//=============================================================================
// ST10_Flow8_FRobot_2.scl
// 1:1 CONVERSION FROM TIA PORTAL V18 GRAPH XML
// Generated: 2026-02-02
//=============================================================================

TYPE
    E_STEP_ST10_Flow8_FRobot_2 : (
        STEP_ST10_Flow8_FRobot_2_WaitRobotScanGripPos2Reach := 304,
        STEP_ST10_Flow8_FRobot_2_S2 := 2,
        STEP_ST10_Flow8_FRobot_2_Step380 := 380,
        STEP_ST10_Flow8_FRobot_2_CodeMove := 248,
        STEP_ST10_Flow8_FRobot_2_F8_Initial := 1,
        STEP_ST10_Flow8_FRobot_2_Maintenance_Pos := 850,
        STEP_ST10_Flow8_FRobot_2_WaitRobotScanGripPos4Reach := 383,
        STEP_ST10_Flow8_FRobot_2_PutPress := 145,
        STEP_ST10_Flow8_FRobot_2_PressGluePickProcessFinish := 549,
        STEP_ST10_Flow8_FRobot_2_WaitRobotScanGripPos3Reach := 372,
        STEP_ST10_Flow8_FRobot_2_DataMove_4 := 262,
        STEP_ST10_Flow8_FRobot_2_Brake_Test := 133,
        STEP_ST10_Flow8_FRobot_2_RobotScanGripPos2Comp := 371,
        STEP_ST10_Flow8_FRobot_2_WaitRobotGripStatus_2 := 366,
        STEP_ST10_Flow8_FRobot_2_S10_InitialFinish := 10,
        STEP_ST10_Flow8_FRobot_2_ScanNGPutFinish_1 := 349,
        STEP_ST10_Flow8_FRobot_2_GluePick := 140,
        STEP_ST10_Flow8_FRobot_2_S8 := 8,
        STEP_ST10_Flow8_FRobot_2_Data_Clear_2 := 258,
        STEP_ST10_Flow8_FRobot_2_WaitRobotFinish_3 := 353,
        STEP_ST10_Flow8_FRobot_2_S5_MESInitial := 5,
        STEP_ST10_Flow8_FRobot_2_DataMove_1 := 255,
        STEP_ST10_Flow8_FRobot_2_PickTableProcess := 400,
        STEP_ST10_Flow8_FRobot_2_StartRobotGlueNGPut := 344,
        STEP_ST10_Flow8_FRobot_2_PartOKStatus_1 := 269,
        STEP_ST10_Flow8_FRobot_2_StartRobotGluePut := 367,
        STEP_ST10_Flow8_FRobot_2_RobotAutoCycle := 329,
        STEP_ST10_Flow8_FRobot_2_BrakeTest_Req := 920,
        STEP_ST10_Flow8_FRobot_2_RobotStart := 316,
        STEP_ST10_Flow8_FRobot_2_GluePut := 155,
        STEP_ST10_Flow8_FRobot_2_PickPallet := 115,
        STEP_ST10_Flow8_FRobot_2_ScanNGPutProcess := 300,
        STEP_ST10_Flow8_FRobot_2_WaitRobot1AndRobot3HomeFinish := 379,
        STEP_ST10_Flow8_FRobot_2_WaitScanCompletely := 247,
        STEP_ST10_Flow8_FRobot_2_WaitRobotGripHaveStatus_3 := 354,
        STEP_ST10_Flow8_FRobot_2_Grip2PartStatus := 244,
        STEP_ST10_Flow8_FRobot_2_GlueNGPutProcess := 350,
        STEP_ST10_Flow8_FRobot_2_ScanMagane := 135,
        STEP_ST10_Flow8_FRobot_2_RobotHome := 317,
        STEP_ST10_Flow8_FRobot_2_WaitRobotGripHaveStatus_2 := 348,
        STEP_ST10_Flow8_FRobot_2_Open_NG_BOX_REQUESTED_ := 111,
        STEP_ST10_Flow8_FRobot_2_RobotScanGripPos4Comp := 391,
        STEP_ST10_Flow8_FRobot_2_Step930 := 930,
        STEP_ST10_Flow8_FRobot_2_ProcessStart := 100,
        STEP_ST10_Flow8_FRobot_2_WaitGripperPos3ScanFinish := 373,
        STEP_ST10_Flow8_FRobot_2_WaitGripperPos1ScanFinish := 296,
        STEP_ST10_Flow8_FRobot_2_WaitGripperPos4ScanFinish := 385,
        STEP_ST10_Flow8_FRobot_2_S_900 := 900,
        STEP_ST10_Flow8_FRobot_2_PartOKStatus := 249,
        STEP_ST10_Flow8_FRobot_2_WaitRobotFinish_1 := 343,
        STEP_ST10_Flow8_FRobot_2_WaitRobotGripStatus_3 := 369,
        STEP_ST10_Flow8_FRobot_2_Grip1PartStatus := 243,
        STEP_ST10_Flow8_FRobot_2_RobotScanGripPos1Comp := 301,
        STEP_ST10_Flow8_FRobot_2_StartRobotPutPress := 361,
        STEP_ST10_Flow8_FRobot_2_WaitRobotHomeRequest := 706,
        STEP_ST10_Flow8_FRobot_2_BrakeTestFinish := 929,
        STEP_ST10_Flow8_FRobot_2_S9 := 9,
        STEP_ST10_Flow8_FRobot_2_Tablecode_Scan := 200,
        STEP_ST10_Flow8_FRobot_2_StartRobotScanNGPut := 328,
        STEP_ST10_Flow8_FRobot_2_ScanMaganeProcess := 450,
        STEP_ST10_Flow8_FRobot_2_StartRobotPickPalletShaft := 326,
        STEP_ST10_Flow8_FRobot_2_WaitRobotFinish_4 := 356,
        STEP_ST10_Flow8_FRobot_2_DataMove_3 := 260,
        STEP_ST10_Flow8_FRobot_2_ScanMaganeProcessFinish := 499,
        STEP_ST10_Flow8_FRobot_2_ScanNGPut := 120,
        STEP_ST10_Flow8_FRobot_2_WaitRobotGripHaveStatus_1 := 347,
        STEP_ST10_Flow8_FRobot_2_DataMove_5 := 264,
        STEP_ST10_Flow8_FRobot_2_MES_Online__offline_ := 384,
        STEP_ST10_Flow8_FRobot_2_WaitRobotFinish_5 := 359,
        STEP_ST10_Flow8_FRobot_2_ScanStart := 246,
        STEP_ST10_Flow8_FRobot_2_PartNGStatus := 251,
        STEP_ST10_Flow8_FRobot_2_Gripe1StatusAlarm := 331,
        STEP_ST10_Flow8_FRobot_2_CheckScanReady := 245,
        STEP_ST10_Flow8_FRobot_2_Gripe2StatusAlarm := 332,
        STEP_ST10_Flow8_FRobot_2_ScanFixtureCode := 110,
        STEP_ST10_Flow8_FRobot_2_WaitRobotGripHaveStatus := 346,
        STEP_ST10_Flow8_FRobot_2_WaitRobotFinish_2 := 345,
        STEP_ST10_Flow8_FRobot_2_PutProcessFinish := 599,
        STEP_ST10_Flow8_FRobot_2_WaitR1HomePosFinsh_1 := 899,
        STEP_ST10_Flow8_FRobot_2_GlueNGPut := 125,
        STEP_ST10_Flow8_FRobot_2_DataMove := 253,
        STEP_ST10_Flow8_FRobot_2_Maintenance := 131,
        STEP_ST10_Flow8_FRobot_2_GluePickProcess := 500,
        STEP_ST10_Flow8_FRobot_2_SetGripCodeScanFlag := 336,
        STEP_ST10_Flow8_FRobot_2_ReqRobotToMantenPos_1 := 704,
        STEP_ST10_Flow8_FRobot_2_WaitRobotReachScanPos := 357,
        STEP_ST10_Flow8_FRobot_2_GlueNGPutFinish := 399,
        STEP_ST10_Flow8_FRobot_2_PickTableProcessFinish := 449,
        STEP_ST10_Flow8_FRobot_2_MasteringTest_Req := 910,
        STEP_ST10_Flow8_FRobot_2_StartRobotScanGripperCode := 338,
        STEP_ST10_Flow8_FRobot_2_RobotScanGripperReachPos1 := 340,
        STEP_ST10_Flow8_FRobot_2_WaitMasteringTestFinish := 911,
        STEP_ST10_Flow8_FRobot_2_WaitRobotGripStatus := 360,
        STEP_ST10_Flow8_FRobot_2_S3 := 3,
        STEP_ST10_Flow8_FRobot_2_PickPalletFinish := 299,
        STEP_ST10_Flow8_FRobot_2_PutPressProcess := 550,
        STEP_ST10_Flow8_FRobot_2_Grip1SensorError := 266,
        STEP_ST10_Flow8_FRobot_2_PressPickProcess := 600,
        STEP_ST10_Flow8_FRobot_2_Data_Clear_6 := 265,
        STEP_ST10_Flow8_FRobot_2_StartRobotScanRing := 355,
        STEP_ST10_Flow8_FRobot_2_WaitRobotFinish := 327,
        STEP_ST10_Flow8_FRobot_2_RobotTaskSelect := 333,
        STEP_ST10_Flow8_FRobot_2_Tablecode_ScanFinish := 149,
        STEP_ST10_Flow8_FRobot_2_GripStatusCheck := 330,
        STEP_ST10_Flow8_FRobot_2_WaitRobotFinish_8 := 368,
        STEP_ST10_Flow8_FRobot_2_WaitRobotFinish_7 := 365,
        STEP_ST10_Flow8_FRobot_2_StartRobotPressPick := 364,
        STEP_ST10_Flow8_FRobot_2_WaitR1MaintenPosFinsh_1 := 705,
        STEP_ST10_Flow8_FRobot_2_PickTable := 130,
        STEP_ST10_Flow8_FRobot_2_RobotReady_ := 311,
        STEP_ST10_Flow8_FRobot_2_Masref_test := 132,
        STEP_ST10_Flow8_FRobot_2_GluePutProcess := 650,
        STEP_ST10_Flow8_FRobot_2_StartRobotGluePick := 358,
        STEP_ST10_Flow8_FRobot_2_PressPickProcessFinish_ := 649,
        STEP_ST10_Flow8_FRobot_2_ReqRobotToHomePos := 707,
        STEP_ST10_Flow8_FRobot_2_DataClear := 252,
        STEP_ST10_Flow8_FRobot_2_StartRobotPickTable := 352,
        STEP_ST10_Flow8_FRobot_2_WaitRobotStartHome := 381,
        STEP_ST10_Flow8_FRobot_2_GluePutProcessFinish := 699,
        STEP_ST10_Flow8_FRobot_2_WaitRobotGripStatus_1 := 363,
        STEP_ST10_Flow8_FRobot_2_WaitRobotFinish_6 := 362,
        STEP_ST10_Flow8_FRobot_2_PickPalletProcess := 250,
        STEP_ST10_Flow8_FRobot_2_RobotSpeed := 4,
        STEP_ST10_Flow8_FRobot_2_RobotManuallyMoved_ := 382,
        STEP_ST10_Flow8_FRobot_2_DataMove_2 := 257,
        STEP_ST10_Flow8_FRobot_2_Grip2SensorError := 267,
        STEP_ST10_Flow8_FRobot_2_WaitBrakeTestFinish := 921,
        STEP_ST10_Flow8_FRobot_2_FlagReset := 268,
        STEP_ST10_Flow8_FRobot_2_PressPick := 150,
        STEP_ST10_Flow8_FRobot_2_WaitGripperPos2ScanFinish := 337,
        STEP_ST10_Flow8_FRobot_2_RobotScanGripPos3Comp := 378,
        STEP_ST10_Flow8_FRobot_2_MasteringTestFinish := 919,
    ) INT := 1;
END_TYPE

CONST
    STEP_ST10_Flow8_FRobot_2_WaitRobotScanGripPos2Reach := 304;
    STEP_ST10_Flow8_FRobot_2_S2 := 2;
    STEP_ST10_Flow8_FRobot_2_Step380 := 380;
    STEP_ST10_Flow8_FRobot_2_CodeMove := 248;
    STEP_ST10_Flow8_FRobot_2_F8_Initial := 1;
    STEP_ST10_Flow8_FRobot_2_Maintenance_Pos := 850;
    STEP_ST10_Flow8_FRobot_2_WaitRobotScanGripPos4Reach := 383;
    STEP_ST10_Flow8_FRobot_2_PutPress := 145;
    STEP_ST10_Flow8_FRobot_2_PressGluePickProcessFinish := 549;
    STEP_ST10_Flow8_FRobot_2_WaitRobotScanGripPos3Reach := 372;
    STEP_ST10_Flow8_FRobot_2_DataMove_4 := 262;
    STEP_ST10_Flow8_FRobot_2_Brake_Test := 133;
    STEP_ST10_Flow8_FRobot_2_RobotScanGripPos2Comp := 371;
    STEP_ST10_Flow8_FRobot_2_WaitRobotGripStatus_2 := 366;
    STEP_ST10_Flow8_FRobot_2_S10_InitialFinish := 10;
    STEP_ST10_Flow8_FRobot_2_ScanNGPutFinish_1 := 349;
    STEP_ST10_Flow8_FRobot_2_GluePick := 140;
    STEP_ST10_Flow8_FRobot_2_S8 := 8;
    STEP_ST10_Flow8_FRobot_2_Data_Clear_2 := 258;
    STEP_ST10_Flow8_FRobot_2_WaitRobotFinish_3 := 353;
    STEP_ST10_Flow8_FRobot_2_S5_MESInitial := 5;
    STEP_ST10_Flow8_FRobot_2_DataMove_1 := 255;
    STEP_ST10_Flow8_FRobot_2_PickTableProcess := 400;
    STEP_ST10_Flow8_FRobot_2_StartRobotGlueNGPut := 344;
    STEP_ST10_Flow8_FRobot_2_PartOKStatus_1 := 269;
    STEP_ST10_Flow8_FRobot_2_StartRobotGluePut := 367;
    STEP_ST10_Flow8_FRobot_2_RobotAutoCycle := 329;
    STEP_ST10_Flow8_FRobot_2_BrakeTest_Req := 920;
    STEP_ST10_Flow8_FRobot_2_RobotStart := 316;
    STEP_ST10_Flow8_FRobot_2_GluePut := 155;
    STEP_ST10_Flow8_FRobot_2_PickPallet := 115;
    STEP_ST10_Flow8_FRobot_2_ScanNGPutProcess := 300;
    STEP_ST10_Flow8_FRobot_2_WaitRobot1AndRobot3HomeFinish := 379;
    STEP_ST10_Flow8_FRobot_2_WaitScanCompletely := 247;
    STEP_ST10_Flow8_FRobot_2_WaitRobotGripHaveStatus_3 := 354;
    STEP_ST10_Flow8_FRobot_2_Grip2PartStatus := 244;
    STEP_ST10_Flow8_FRobot_2_GlueNGPutProcess := 350;
    STEP_ST10_Flow8_FRobot_2_ScanMagane := 135;
    STEP_ST10_Flow8_FRobot_2_RobotHome := 317;
    STEP_ST10_Flow8_FRobot_2_WaitRobotGripHaveStatus_2 := 348;
    STEP_ST10_Flow8_FRobot_2_Open_NG_BOX_REQUESTED_ := 111;
    STEP_ST10_Flow8_FRobot_2_RobotScanGripPos4Comp := 391;
    STEP_ST10_Flow8_FRobot_2_Step930 := 930;
    STEP_ST10_Flow8_FRobot_2_ProcessStart := 100;
    STEP_ST10_Flow8_FRobot_2_WaitGripperPos3ScanFinish := 373;
    STEP_ST10_Flow8_FRobot_2_WaitGripperPos1ScanFinish := 296;
    STEP_ST10_Flow8_FRobot_2_WaitGripperPos4ScanFinish := 385;
    STEP_ST10_Flow8_FRobot_2_S_900 := 900;
    STEP_ST10_Flow8_FRobot_2_PartOKStatus := 249;
    STEP_ST10_Flow8_FRobot_2_WaitRobotFinish_1 := 343;
    STEP_ST10_Flow8_FRobot_2_WaitRobotGripStatus_3 := 369;
    STEP_ST10_Flow8_FRobot_2_Grip1PartStatus := 243;
    STEP_ST10_Flow8_FRobot_2_RobotScanGripPos1Comp := 301;
    STEP_ST10_Flow8_FRobot_2_StartRobotPutPress := 361;
    STEP_ST10_Flow8_FRobot_2_WaitRobotHomeRequest := 706;
    STEP_ST10_Flow8_FRobot_2_BrakeTestFinish := 929;
    STEP_ST10_Flow8_FRobot_2_S9 := 9;
    STEP_ST10_Flow8_FRobot_2_Tablecode_Scan := 200;
    STEP_ST10_Flow8_FRobot_2_StartRobotScanNGPut := 328;
    STEP_ST10_Flow8_FRobot_2_ScanMaganeProcess := 450;
    STEP_ST10_Flow8_FRobot_2_StartRobotPickPalletShaft := 326;
    STEP_ST10_Flow8_FRobot_2_WaitRobotFinish_4 := 356;
    STEP_ST10_Flow8_FRobot_2_DataMove_3 := 260;
    STEP_ST10_Flow8_FRobot_2_ScanMaganeProcessFinish := 499;
    STEP_ST10_Flow8_FRobot_2_ScanNGPut := 120;
    STEP_ST10_Flow8_FRobot_2_WaitRobotGripHaveStatus_1 := 347;
    STEP_ST10_Flow8_FRobot_2_DataMove_5 := 264;
    STEP_ST10_Flow8_FRobot_2_MES_Online__offline_ := 384;
    STEP_ST10_Flow8_FRobot_2_WaitRobotFinish_5 := 359;
    STEP_ST10_Flow8_FRobot_2_ScanStart := 246;
    STEP_ST10_Flow8_FRobot_2_PartNGStatus := 251;
    STEP_ST10_Flow8_FRobot_2_Gripe1StatusAlarm := 331;
    STEP_ST10_Flow8_FRobot_2_CheckScanReady := 245;
    STEP_ST10_Flow8_FRobot_2_Gripe2StatusAlarm := 332;
    STEP_ST10_Flow8_FRobot_2_ScanFixtureCode := 110;
    STEP_ST10_Flow8_FRobot_2_WaitRobotGripHaveStatus := 346;
    STEP_ST10_Flow8_FRobot_2_WaitRobotFinish_2 := 345;
    STEP_ST10_Flow8_FRobot_2_PutProcessFinish := 599;
    STEP_ST10_Flow8_FRobot_2_WaitR1HomePosFinsh_1 := 899;
    STEP_ST10_Flow8_FRobot_2_GlueNGPut := 125;
    STEP_ST10_Flow8_FRobot_2_DataMove := 253;
    STEP_ST10_Flow8_FRobot_2_Maintenance := 131;
    STEP_ST10_Flow8_FRobot_2_GluePickProcess := 500;
    STEP_ST10_Flow8_FRobot_2_SetGripCodeScanFlag := 336;
    STEP_ST10_Flow8_FRobot_2_ReqRobotToMantenPos_1 := 704;
    STEP_ST10_Flow8_FRobot_2_WaitRobotReachScanPos := 357;
    STEP_ST10_Flow8_FRobot_2_GlueNGPutFinish := 399;
    STEP_ST10_Flow8_FRobot_2_PickTableProcessFinish := 449;
    STEP_ST10_Flow8_FRobot_2_MasteringTest_Req := 910;
    STEP_ST10_Flow8_FRobot_2_StartRobotScanGripperCode := 338;
    STEP_ST10_Flow8_FRobot_2_RobotScanGripperReachPos1 := 340;
    STEP_ST10_Flow8_FRobot_2_WaitMasteringTestFinish := 911;
    STEP_ST10_Flow8_FRobot_2_WaitRobotGripStatus := 360;
    STEP_ST10_Flow8_FRobot_2_S3 := 3;
    STEP_ST10_Flow8_FRobot_2_PickPalletFinish := 299;
    STEP_ST10_Flow8_FRobot_2_PutPressProcess := 550;
    STEP_ST10_Flow8_FRobot_2_Grip1SensorError := 266;
    STEP_ST10_Flow8_FRobot_2_PressPickProcess := 600;
    STEP_ST10_Flow8_FRobot_2_Data_Clear_6 := 265;
    STEP_ST10_Flow8_FRobot_2_StartRobotScanRing := 355;
    STEP_ST10_Flow8_FRobot_2_WaitRobotFinish := 327;
    STEP_ST10_Flow8_FRobot_2_RobotTaskSelect := 333;
    STEP_ST10_Flow8_FRobot_2_Tablecode_ScanFinish := 149;
    STEP_ST10_Flow8_FRobot_2_GripStatusCheck := 330;
    STEP_ST10_Flow8_FRobot_2_WaitRobotFinish_8 := 368;
    STEP_ST10_Flow8_FRobot_2_WaitRobotFinish_7 := 365;
    STEP_ST10_Flow8_FRobot_2_StartRobotPressPick := 364;
    STEP_ST10_Flow8_FRobot_2_WaitR1MaintenPosFinsh_1 := 705;
    STEP_ST10_Flow8_FRobot_2_PickTable := 130;
    STEP_ST10_Flow8_FRobot_2_RobotReady_ := 311;
    STEP_ST10_Flow8_FRobot_2_Masref_test := 132;
    STEP_ST10_Flow8_FRobot_2_GluePutProcess := 650;
    STEP_ST10_Flow8_FRobot_2_StartRobotGluePick := 358;
    STEP_ST10_Flow8_FRobot_2_PressPickProcessFinish_ := 649;
    STEP_ST10_Flow8_FRobot_2_ReqRobotToHomePos := 707;
    STEP_ST10_Flow8_FRobot_2_DataClear := 252;
    STEP_ST10_Flow8_FRobot_2_StartRobotPickTable := 352;
    STEP_ST10_Flow8_FRobot_2_WaitRobotStartHome := 381;
    STEP_ST10_Flow8_FRobot_2_GluePutProcessFinish := 699;
    STEP_ST10_Flow8_FRobot_2_WaitRobotGripStatus_1 := 363;
    STEP_ST10_Flow8_FRobot_2_WaitRobotFinish_6 := 362;
    STEP_ST10_Flow8_FRobot_2_PickPalletProcess := 250;
    STEP_ST10_Flow8_FRobot_2_RobotSpeed := 4;
    STEP_ST10_Flow8_FRobot_2_RobotManuallyMoved_ := 382;
    STEP_ST10_Flow8_FRobot_2_DataMove_2 := 257;
    STEP_ST10_Flow8_FRobot_2_Grip2SensorError := 267;
    STEP_ST10_Flow8_FRobot_2_WaitBrakeTestFinish := 921;
    STEP_ST10_Flow8_FRobot_2_FlagReset := 268;
    STEP_ST10_Flow8_FRobot_2_PressPick := 150;
    STEP_ST10_Flow8_FRobot_2_WaitGripperPos2ScanFinish := 337;
    STEP_ST10_Flow8_FRobot_2_RobotScanGripPos3Comp := 378;
    STEP_ST10_Flow8_FRobot_2_MasteringTestFinish := 919;
END_CONST

FUNCTION_BLOCK "ST10_Flow8_FRobot_2_1to1"
{ S7_Optimized_Access := 'TRUE' }
VERSION : 1.0

VAR_INPUT
    iSysInface : "RCS_SysComInterface_V1";
END_VAR

VAR_IN_OUT
    ioPM_Inface : "RCS_PMInterface_V1";
    ioStatus : Int;
END_VAR

VAR_OUTPUT
    oAlarmID : Int;
END_VAR

VAR
    State : INT := 1;
    act_InitialRun : Bool;
    act_InitialOK : Bool;
    act_WaitRunning : Bool;
    act_Running : Bool;
    act_ProcessComplete : Bool;
    act_ProcessStart : Bool;
    act_UnPause : Bool;
    bError : Bool;
    wErrorID : Word;
END_VAR

BEGIN
    //======================================================================
    // STATE MACHINE - Inline Transition Conditions
    //======================================================================

    CASE #State OF

        // ===========================================
        // STEP 304: WaitRobotScanGripPos2Reach
        // ===========================================
        STEP_ST10_Flow8_FRobot_2_WaitRobotScanGripPos2Reach:
            // No actions in XML

            // Transition to next step: 2
            IF TRUE THEN  // Sequential transition - review XML for actual condition
                #State := STEP_ST10_Flow8_FRobot_2_S2;
            END_IF;

        // ===========================================
        // STEP 2: S2
        // ===========================================
        STEP_ST10_Flow8_FRobot_2_S2:
            // No actions in XML

            // Transition to next step: 380
            IF TRUE THEN  // Sequential transition - review XML for actual condition
                #State := STEP_ST10_Flow8_FRobot_2_Step380;
            END_IF;

        // ===========================================
        // STEP 380: Step380
        // ===========================================
        STEP_ST10_Flow8_FRobot_2_Step380:
            // No actions in XML

            // Transition to next step: 248
            IF TRUE THEN  // Sequential transition - review XML for actual condition
                #State := STEP_ST10_Flow8_FRobot_2_CodeMove;
            END_IF;

        // ===========================================
        // STEP 248: CodeMove
        // ===========================================
        STEP_ST10_Flow8_FRobot_2_CodeMove:
            // Action Qualifier=N
            // Token: "AutoProcessData".F_Robot2Grip2.Code_1 := "KeyenceSR1000Ctrl_806A1DB".sHMI.Status.CurrentCode
            "AutoProcessData".F_Robot2Grip2.Code_1 := "KeyenceSR1000Ctrl_806A1DB".sHMI.Status.CurrentCode;

            // Transition to next step: 1
            IF TRUE THEN  // Sequential transition - review XML for actual condition
                #State := STEP_ST10_Flow8_FRobot_2_F8_Initial;
            END_IF;

        // ===========================================
        // STEP 1: F8_Initial
        // ===========================================
        STEP_ST10_Flow8_FRobot_2_F8_Initial:
            // Action Qualifier=S
            // Token: #ioPM_Inface.InitialRun
            #ioPM_Inface.InitialRun := TRUE;
            // Action Qualifier=R
            // Token: #ioPM_Inface.InitialOK
            #ioPM_Inface.InitialOK := FALSE;
            // Action Qualifier=R
            // Token: #ioPM_Inface.WaitRunning
            #ioPM_Inface.WaitRunning := FALSE;
            // Action Qualifier=R
            // Token: #ioPM_Inface.Running
            #ioPM_Inface.Running := FALSE;
            // Action Qualifier=R
            // Token: #ioPM_Inface.UnPause
            #ioPM_Inface.UnPause := FALSE;
            // Action Qualifier=R
            // Token: "Station_Sys".Cmd.Calibration
            "Station_Sys".Cmd.Calibration := FALSE;
            // Action Qualifier=R
            // Token: "Station_Sys".Cmd.ChangeOver
            "Station_Sys".Cmd.ChangeOver := FALSE;
            // Action Qualifier=N
            // Token: //"ST350_Sys".Cmd.DryRun
            //"ST350_Sys".Cmd.DryRun;
            // Action Qualifier=R
            // Token: "Station_Sys".Cmd.Reserve
            "Station_Sys".Cmd.Reserve := FALSE;
            // Action Qualifier=R
            // Token: "Station_Sys".Cmd.OneCycle
            "Station_Sys".Cmd.OneCycle := FALSE;
            // Action Qualifier=R
            // Token: "AutoProcessControl".Robot_2.PalletPickFlag
            "AutoProcessControl".Robot_2.PalletPickFlag := FALSE;
            // Action Qualifier=R
            // Token: "AutoProcessControl".Robot_2.MagnetScanFlag
            "AutoProcessControl".Robot_2.MagnetScanFlag := FALSE;
            // Action Qualifier=R
            // Token: "AutoProcessControl".Robot_2.GluePutFlag
            "AutoProcessControl".Robot_2.GluePutFlag := FALSE;
            // Action Qualifier=R
            // Token: "AutoProcessControl".Robot_2.GluePickFlag
            "AutoProcessControl".Robot_2.GluePickFlag := FALSE;
            // Action Qualifier=R
            // Token: "AutoProcessControl".Robot_2.Press2PutFlag
            "AutoProcessControl".Robot_2.Press2PutFlag := FALSE;
            // Action Qualifier=R
            // Token: "AutoProcessControl".Robot_2.GlueNGPutFlag
            "AutoProcessControl".Robot_2.GlueNGPutFlag := FALSE;
            // Action Qualifier=R
            // Token: "AutoProcessControl".Robot_2.ScanNGPutFlag
            "AutoProcessControl".Robot_2.ScanNGPutFlag := FALSE;
            // Action Qualifier=R
            // Token: #ioPM_Inface.ProcessComplete
            #ioPM_Inface.ProcessComplete := FALSE;
            // Action Qualifier=R
            // Token: #ioPM_Inface.ProcessStart
            #ioPM_Inface.ProcessStart := FALSE;
            // Action Qualifier=R
            // Token: "ChangeOver_DB".Robot_2.MaintenancePosReqSelFlag
            "ChangeOver_DB".Robot_2.MaintenancePosReqSelFlag := FALSE;
            // Action Qualifier=N
            // Token: //"Robot_DB".Robot_2.MasteringTest_Req
            //"Robot_DB".Robot_2.MasteringTest_Req;
            // Action Qualifier=N
            // Token: //"Robot_DB".Robot_2.BrakeTest_Req
            //"Robot_DB".Robot_2.BrakeTest_Req;
            // Action Qualifier=R
            // Token: #Auto_Run_after_NG_box_closed
            #Auto_Run_after_NG_box_closed := FALSE;

            // Transition to next step: 850
            IF TRUE THEN  // Sequential transition - review XML for actual condition
                #State := STEP_ST10_Flow8_FRobot_2_Maintenance_Pos;
            END_IF;

        // ===========================================
        // STEP 850: Maintenance Pos
        // ===========================================
        STEP_ST10_Flow8_FRobot_2_Maintenance_Pos:
            // No actions in XML

            // Transition to next step: 383
            IF TRUE THEN  // Sequential transition - review XML for actual condition
                #State := STEP_ST10_Flow8_FRobot_2_WaitRobotScanGripPos4Reach;
            END_IF;

        // ===========================================
        // STEP 383: WaitRobotScanGripPos4Reach
        // ===========================================
        STEP_ST10_Flow8_FRobot_2_WaitRobotScanGripPos4Reach:
            // No actions in XML

            // Transition to next step: 145
            IF TRUE THEN  // Sequential transition - review XML for actual condition
                #State := STEP_ST10_Flow8_FRobot_2_PutPress;
            END_IF;

        // ===========================================
        // STEP 145: PutPress
        // ===========================================
        STEP_ST10_Flow8_FRobot_2_PutPress:
            // Action Qualifier=S
            // Token: "AutoProcessControl".Robot_2.Press2PutFlag
            "AutoProcessControl".Robot_2.Press2PutFlag := TRUE;
            // Action Qualifier=R
            // Token: #ioPM_Inface.ProcessComplete
            #ioPM_Inface.ProcessComplete := FALSE;
            // Action Qualifier=S
            // Token: #ioPM_Inface.ProcessStart
            #ioPM_Inface.ProcessStart := TRUE;

            // Transition to next step: 549
            IF TRUE THEN  // Sequential transition - review XML for actual condition
                #State := STEP_ST10_Flow8_FRobot_2_PressGluePickProcessFinish;
            END_IF;

        // ===========================================
        // STEP 549: PressGluePickProcessFinish
        // ===========================================
        STEP_ST10_Flow8_FRobot_2_PressGluePickProcessFinish:
            // Action Qualifier=S
            // Token: #ioPM_Inface.ProcessComplete
            #ioPM_Inface.ProcessComplete := TRUE;
            // Action Qualifier=R
            // Token: #ioPM_Inface.ProcessStart
            #ioPM_Inface.ProcessStart := FALSE;

            // Transition to next step: 372
            IF TRUE THEN  // Sequential transition - review XML for actual condition
                #State := STEP_ST10_Flow8_FRobot_2_WaitRobotScanGripPos3Reach;
            END_IF;

        // ===========================================
        // STEP 372: WaitRobotScanGripPos3Reach
        // ===========================================
        STEP_ST10_Flow8_FRobot_2_WaitRobotScanGripPos3Reach:
            // No actions in XML

            // Transition to next step: 262
            IF TRUE THEN  // Sequential transition - review XML for actual condition
                #State := STEP_ST10_Flow8_FRobot_2_DataMove_4;
            END_IF;

        // ===========================================
        // STEP 262: DataMove_4
        // ===========================================
        STEP_ST10_Flow8_FRobot_2_DataMove_4:
            // Action Qualifier=N, Event="S1"
            // Token: "AutoProcessData".F_Robot2Grip1 := "AutoProcessData".B_Press1
            "AutoProcessData".F_Robot2Grip1 := "AutoProcessData".B_Press1;
            // Action Qualifier=N, Event="S1"
            // Token: "AutoProcessData".B_Press1 := "AutoProcessData".ClearData
            "AutoProcessData".B_Press1 := "AutoProcessData".ClearData;

            // Transition to next step: 133
            IF TRUE THEN  // Sequential transition - review XML for actual condition
                #State := STEP_ST10_Flow8_FRobot_2_Brake_Test;
            END_IF;

        // ===========================================
        // STEP 133: Brake_Test
        // ===========================================
        STEP_ST10_Flow8_FRobot_2_Brake_Test:
            // Action Qualifier=R
            // Token: #ioPM_Inface.ProcessComplete
            #ioPM_Inface.ProcessComplete := FALSE;
            // Action Qualifier=S
            // Token: #ioPM_Inface.ProcessStart
            #ioPM_Inface.ProcessStart := TRUE;

            // Transition to next step: 371
            IF TRUE THEN  // Sequential transition - review XML for actual condition
                #State := STEP_ST10_Flow8_FRobot_2_RobotScanGripPos2Comp;
            END_IF;

        // ===========================================
        // STEP 371: RobotScanGripPos2Comp
        // ===========================================
        STEP_ST10_Flow8_FRobot_2_RobotScanGripPos2Comp:
            // No actions in XML

            // Transition to next step: 366
            IF TRUE THEN  // Sequential transition - review XML for actual condition
                #State := STEP_ST10_Flow8_FRobot_2_WaitRobotGripStatus_2;
            END_IF;

        // ===========================================
        // STEP 366: WaitRobotGripStatus_2
        // ===========================================
        STEP_ST10_Flow8_FRobot_2_WaitRobotGripStatus_2:
            // No actions in XML

            // Transition to next step: 10
            IF TRUE THEN  // Sequential transition - review XML for actual condition
                #State := STEP_ST10_Flow8_FRobot_2_S10_InitialFinish;
            END_IF;

        // ===========================================
        // STEP 10: S10_InitialFinish
        // ===========================================
        STEP_ST10_Flow8_FRobot_2_S10_InitialFinish:
            // Action Qualifier=S
            // Token: #ioPM_Inface.InitialOK
            #ioPM_Inface.InitialOK := TRUE;

            // Transition to next step: 349
            IF TRUE THEN  // Sequential transition - review XML for actual condition
                #State := STEP_ST10_Flow8_FRobot_2_ScanNGPutFinish_1;
            END_IF;

        // ===========================================
        // STEP 349: ScanNGPutFinish_1
        // ===========================================
        STEP_ST10_Flow8_FRobot_2_ScanNGPutFinish_1:
            // Action Qualifier=S
            // Token: #ioPM_Inface.ProcessComplete
            #ioPM_Inface.ProcessComplete := TRUE;
            // Action Qualifier=R
            // Token: #ioPM_Inface.ProcessStart
            #ioPM_Inface.ProcessStart := FALSE;

            // Transition to next step: 140
            IF TRUE THEN  // Sequential transition - review XML for actual condition
                #State := STEP_ST10_Flow8_FRobot_2_GluePick;
            END_IF;

        // ===========================================
        // STEP 140: GluePick
        // ===========================================
        STEP_ST10_Flow8_FRobot_2_GluePick:
            // Action Qualifier=S
            // Token: "AutoProcessControl".Robot_2.GluePickFlag
            "AutoProcessControl".Robot_2.GluePickFlag := TRUE;
            // Action Qualifier=R
            // Token: #ioPM_Inface.ProcessComplete
            #ioPM_Inface.ProcessComplete := FALSE;
            // Action Qualifier=S
            // Token: #ioPM_Inface.ProcessStart
            #ioPM_Inface.ProcessStart := TRUE;

            // Transition to next step: 8
            IF TRUE THEN  // Sequential transition - review XML for actual condition
                #State := STEP_ST10_Flow8_FRobot_2_S8;
            END_IF;

        // ===========================================
        // STEP 8: S8
        // ===========================================
        STEP_ST10_Flow8_FRobot_2_S8:
            // No actions in XML

            // Transition to next step: 258
            IF TRUE THEN  // Sequential transition - review XML for actual condition
                #State := STEP_ST10_Flow8_FRobot_2_Data_Clear_2;
            END_IF;

        // ===========================================
        // STEP 258: Data Clear_2
        // ===========================================
        STEP_ST10_Flow8_FRobot_2_Data_Clear_2:
            // Action Qualifier=N, Event="S1"
            // Token: "AutoProcessData".F_Robot2Grip2 := "AutoProcessData".ClearData
            "AutoProcessData".F_Robot2Grip2 := "AutoProcessData".ClearData;

            // Transition to next step: 353
            IF TRUE THEN  // Sequential transition - review XML for actual condition
                #State := STEP_ST10_Flow8_FRobot_2_WaitRobotFinish_3;
            END_IF;

        // ===========================================
        // STEP 353: WaitRobotFinish_3
        // ===========================================
        STEP_ST10_Flow8_FRobot_2_WaitRobotFinish_3:
            // No actions in XML

            // Transition to next step: 5
            IF TRUE THEN  // Sequential transition - review XML for actual condition
                #State := STEP_ST10_Flow8_FRobot_2_S5_MESInitial;
            END_IF;

        // ===========================================
        // STEP 5: S5_MESInitial
        // ===========================================
        STEP_ST10_Flow8_FRobot_2_S5_MESInitial:
            // No actions in XML

            // Transition to next step: 255
            IF TRUE THEN  // Sequential transition - review XML for actual condition
                #State := STEP_ST10_Flow8_FRobot_2_DataMove_1;
            END_IF;

        // ===========================================
        // STEP 255: DataMove_1
        // ===========================================
        STEP_ST10_Flow8_FRobot_2_DataMove_1:
            // Action Qualifier=N, Event="S1"
            // Token: "AutoProcessData".C_GlueNGBuffer := "AutoProcessData".F_Robot2Grip1
            "AutoProcessData".C_GlueNGBuffer := "AutoProcessData".F_Robot2Grip1;
            // Action Qualifier=N, Event="S1"
            // Token: "AutoProcessData".F_Robot2Grip1 := "AutoProcessData".ClearData
            "AutoProcessData".F_Robot2Grip1 := "AutoProcessData".ClearData;

            // Transition to next step: 400
            IF TRUE THEN  // Sequential transition - review XML for actual condition
                #State := STEP_ST10_Flow8_FRobot_2_PickTableProcess;
            END_IF;

        // ===========================================
        // STEP 400: PickTableProcess
        // ===========================================
        STEP_ST10_Flow8_FRobot_2_PickTableProcess:
            // No actions in XML

            // Transition to next step: 344
            IF TRUE THEN  // Sequential transition - review XML for actual condition
                #State := STEP_ST10_Flow8_FRobot_2_StartRobotGlueNGPut;
            END_IF;

        // ===========================================
        // STEP 344: StartRobotGlueNGPut
        // ===========================================
        STEP_ST10_Flow8_FRobot_2_StartRobotGlueNGPut:
            // Action Qualifier=N
            // Token: "KukaRobot2_CtrlDB".sPLCtoROB.User.Cycle.DI253_GlueNGPutReq
            "KukaRobot2_CtrlDB".sPLCtoROB.User.Cycle.DI253_GlueNGPutReq;

            // Transition to next step: 269
            IF TRUE THEN  // Sequential transition - review XML for actual condition
                #State := STEP_ST10_Flow8_FRobot_2_PartOKStatus_1;
            END_IF;

        // ===========================================
        // STEP 269: PartOKStatus_1
        // ===========================================
        STEP_ST10_Flow8_FRobot_2_PartOKStatus_1:
            // Action Qualifier=N
            // Token: "AutoProcessData".F_Robot2Grip2.PartStatus := 110
            "AutoProcessData".F_Robot2Grip2.PartStatus := 110;

            // Transition to next step: 367
            IF TRUE THEN  // Sequential transition - review XML for actual condition
                #State := STEP_ST10_Flow8_FRobot_2_StartRobotGluePut;
            END_IF;

        // ===========================================
        // STEP 367: StartRobotGluePut
        // ===========================================
        STEP_ST10_Flow8_FRobot_2_StartRobotGluePut:
            // Action Qualifier=N
            // Token: "KukaRobot2_CtrlDB".sPLCtoROB.User.Cycle.DI265_GluePutReq
            "KukaRobot2_CtrlDB".sPLCtoROB.User.Cycle.DI265_GluePutReq;

            // Transition to next step: 329
            IF TRUE THEN  // Sequential transition - review XML for actual condition
                #State := STEP_ST10_Flow8_FRobot_2_RobotAutoCycle;
            END_IF;

        // ===========================================
        // STEP 329: RobotAutoCycle
        // ===========================================
        STEP_ST10_Flow8_FRobot_2_RobotAutoCycle:
            // Action Qualifier=N
            // Token: "KukaRobot2_CtrlDB".ioStartAutoCycle
            "KukaRobot2_CtrlDB".ioStartAutoCycle;

            // Transition to next step: 920
            IF TRUE THEN  // Sequential transition - review XML for actual condition
                #State := STEP_ST10_Flow8_FRobot_2_BrakeTest_Req;
            END_IF;

        // ===========================================
        // STEP 920: BrakeTest_Req
        // ===========================================
        STEP_ST10_Flow8_FRobot_2_BrakeTest_Req:
            // Action Qualifier=N
            // Token: "KukaRobot2_CtrlDB".sPLCtoROB.User.Cycle.DI329
            "KukaRobot2_CtrlDB".sPLCtoROB.User.Cycle.DI329;
            // Action Qualifier=N
            // Token: "KukaRobot2_CtrlDB".sPLCtoROB.User.Safety.DI451
            "KukaRobot2_CtrlDB".sPLCtoROB.User.Safety.DI451;

            // Transition to next step: 316
            IF TRUE THEN  // Sequential transition - review XML for actual condition
                #State := STEP_ST10_Flow8_FRobot_2_RobotStart;
            END_IF;

        // ===========================================
        // STEP 316: RobotStart
        // ===========================================
        STEP_ST10_Flow8_FRobot_2_RobotStart:
            // Action Qualifier=N
            // Token: "KukaRobot2_CtrlDB".ioAutoStart
            "KukaRobot2_CtrlDB".ioAutoStart;

            // Transition to next step: 155
            IF TRUE THEN  // Sequential transition - review XML for actual condition
                #State := STEP_ST10_Flow8_FRobot_2_GluePut;
            END_IF;

        // ===========================================
        // STEP 155: GluePut
        // ===========================================
        STEP_ST10_Flow8_FRobot_2_GluePut:
            // Action Qualifier=S
            // Token: "AutoProcessControl".Robot_2.GluePutFlag
            "AutoProcessControl".Robot_2.GluePutFlag := TRUE;
            // Action Qualifier=R
            // Token: #ioPM_Inface.ProcessComplete
            #ioPM_Inface.ProcessComplete := FALSE;
            // Action Qualifier=S
            // Token: #ioPM_Inface.ProcessStart
            #ioPM_Inface.ProcessStart := TRUE;

            // Transition to next step: 115
            IF TRUE THEN  // Sequential transition - review XML for actual condition
                #State := STEP_ST10_Flow8_FRobot_2_PickPallet;
            END_IF;

        // ===========================================
        // STEP 115: PickPallet
        // ===========================================
        STEP_ST10_Flow8_FRobot_2_PickPallet:
            // Action Qualifier=S
            // Token: "AutoProcessControl".Robot_2.PalletPickFlag
            "AutoProcessControl".Robot_2.PalletPickFlag := TRUE;
            // Action Qualifier=R
            // Token: #ioPM_Inface.ProcessComplete
            #ioPM_Inface.ProcessComplete := FALSE;
            // Action Qualifier=S
            // Token: #ioPM_Inface.ProcessStart
            #ioPM_Inface.ProcessStart := TRUE;

            // Transition to next step: 300
            IF TRUE THEN  // Sequential transition - review XML for actual condition
                #State := STEP_ST10_Flow8_FRobot_2_ScanNGPutProcess;
            END_IF;

        // ===========================================
        // STEP 300: ScanNGPutProcess
        // ===========================================
        STEP_ST10_Flow8_FRobot_2_ScanNGPutProcess:
            // No actions in XML

            // Transition to next step: 379
            IF TRUE THEN  // Sequential transition - review XML for actual condition
                #State := STEP_ST10_Flow8_FRobot_2_WaitRobot1AndRobot3HomeFinish;
            END_IF;

        // ===========================================
        // STEP 379: WaitRobot1AndRobot3HomeFinish
        // ===========================================
        STEP_ST10_Flow8_FRobot_2_WaitRobot1AndRobot3HomeFinish:
            // No actions in XML

            // Transition to next step: 247
            IF TRUE THEN  // Sequential transition - review XML for actual condition
                #State := STEP_ST10_Flow8_FRobot_2_WaitScanCompletely;
            END_IF;

        // ===========================================
        // STEP 247: WaitScanCompletely
        // ===========================================
        STEP_ST10_Flow8_FRobot_2_WaitScanCompletely:
            // No actions in XML

            // Transition to next step: 354
            IF TRUE THEN  // Sequential transition - review XML for actual condition
                #State := STEP_ST10_Flow8_FRobot_2_WaitRobotGripHaveStatus_3;
            END_IF;

        // ===========================================
        // STEP 354: WaitRobotGripHaveStatus_3
        // ===========================================
        STEP_ST10_Flow8_FRobot_2_WaitRobotGripHaveStatus_3:
            // No actions in XML

            // Transition to next step: 244
            IF TRUE THEN  // Sequential transition - review XML for actual condition
                #State := STEP_ST10_Flow8_FRobot_2_Grip2PartStatus;
            END_IF;

        // ===========================================
        // STEP 244: Grip2PartStatus
        // ===========================================
        STEP_ST10_Flow8_FRobot_2_Grip2PartStatus:
            // Action Qualifier=N
            // Token: "AutoProcessData".F_Robot2Grip2.PartStatus := 100
            "AutoProcessData".F_Robot2Grip2.PartStatus := 100;

            // Transition to next step: 350
            IF TRUE THEN  // Sequential transition - review XML for actual condition
                #State := STEP_ST10_Flow8_FRobot_2_GlueNGPutProcess;
            END_IF;

        // ===========================================
        // STEP 350: GlueNGPutProcess
        // ===========================================
        STEP_ST10_Flow8_FRobot_2_GlueNGPutProcess:
            // No actions in XML

            // Transition to next step: 135
            IF TRUE THEN  // Sequential transition - review XML for actual condition
                #State := STEP_ST10_Flow8_FRobot_2_ScanMagane;
            END_IF;

        // ===========================================
        // STEP 135: ScanMagane
        // ===========================================
        STEP_ST10_Flow8_FRobot_2_ScanMagane:
            // Action Qualifier=S
            // Token: "AutoProcessControl".Robot_2.MagnetScanFlag
            "AutoProcessControl".Robot_2.MagnetScanFlag := TRUE;
            // Action Qualifier=R
            // Token: #ioPM_Inface.ProcessComplete
            #ioPM_Inface.ProcessComplete := FALSE;
            // Action Qualifier=S
            // Token: #ioPM_Inface.ProcessStart
            #ioPM_Inface.ProcessStart := TRUE;

            // Transition to next step: 317
            IF TRUE THEN  // Sequential transition - review XML for actual condition
                #State := STEP_ST10_Flow8_FRobot_2_RobotHome;
            END_IF;

        // ===========================================
        // STEP 317: RobotHome
        // ===========================================
        STEP_ST10_Flow8_FRobot_2_RobotHome:
            // Action Qualifier=N
            // Token: "KukaRobot2_CtrlDB".ioSrartHome
            "KukaRobot2_CtrlDB".ioSrartHome;

            // Transition to next step: 348
            IF TRUE THEN  // Sequential transition - review XML for actual condition
                #State := STEP_ST10_Flow8_FRobot_2_WaitRobotGripHaveStatus_2;
            END_IF;

        // ===========================================
        // STEP 348: WaitRobotGripHaveStatus_2
        // ===========================================
        STEP_ST10_Flow8_FRobot_2_WaitRobotGripHaveStatus_2:
            // No actions in XML

            // Transition to next step: 111
            IF TRUE THEN  // Sequential transition - review XML for actual condition
                #State := STEP_ST10_Flow8_FRobot_2_Open_NG_BOX_REQUESTED_;
            END_IF;

        // ===========================================
        // STEP 111: Open NG BOX REQUESTED?
        // ===========================================
        STEP_ST10_Flow8_FRobot_2_Open_NG_BOX_REQUESTED_:
            // No actions in XML

            // Transition to next step: 391
            IF TRUE THEN  // Sequential transition - review XML for actual condition
                #State := STEP_ST10_Flow8_FRobot_2_RobotScanGripPos4Comp;
            END_IF;

        // ===========================================
        // STEP 391: RobotScanGripPos4Comp
        // ===========================================
        STEP_ST10_Flow8_FRobot_2_RobotScanGripPos4Comp:
            // Action Qualifier=N
            // Token: "KukaRobot2_CtrlDB".sPLCtoROB.User.Cycle.DI307_ScanPartFinish
            "KukaRobot2_CtrlDB".sPLCtoROB.User.Cycle.DI307_ScanPartFinish;
            // Action Qualifier=N
            // Token: "KukaRobot2_CtrlDB".sPLCtoROB.User.Cycle.DI306_ScanPartComplete
            "KukaRobot2_CtrlDB".sPLCtoROB.User.Cycle.DI306_ScanPartComplete;

            // Transition to next step: 930
            IF TRUE THEN  // Sequential transition - review XML for actual condition
                #State := STEP_ST10_Flow8_FRobot_2_Step930;
            END_IF;

        // ===========================================
        // STEP 930: Step930
        // ===========================================
        STEP_ST10_Flow8_FRobot_2_Step930:
            // Action Qualifier=N
            // Token: "AutoProcessData".C_MagnScanNGBuffer.PartStatus := 0
            "AutoProcessData".C_MagnScanNGBuffer.PartStatus := 0;

            // Transition to next step: 100
            IF TRUE THEN  // Sequential transition - review XML for actual condition
                #State := STEP_ST10_Flow8_FRobot_2_ProcessStart;
            END_IF;

        // ===========================================
        // STEP 100: ProcessStart
        // ===========================================
        STEP_ST10_Flow8_FRobot_2_ProcessStart:
            // Action Qualifier=R
            // Token: #ioPM_Inface.InitialRun
            #ioPM_Inface.InitialRun := FALSE;
            // Action Qualifier=R
            // Token: #ioPM_Inface.ProcessComplete
            #ioPM_Inface.ProcessComplete := FALSE;
            // Action Qualifier=R
            // Token: #ioPM_Inface.ProcessStart
            #ioPM_Inface.ProcessStart := FALSE;
            // Action Qualifier=S
            // Token: #ioPM_Inface.InitialOK
            #ioPM_Inface.InitialOK := TRUE;
            // Action Qualifier=S
            // Token: #ioPM_Inface.WaitRunning
            #ioPM_Inface.WaitRunning := TRUE;
            // Action Qualifier=N, Event="S1"
            // Token: #ioPM_Inface.ProcessResult := 0
            #ioPM_Inface.ProcessResult := 0;
            // Action Qualifier=R
            // Token: "ST10_GeneralData".FlowControl_Handshake[8].Start
            "ST10_GeneralData".FlowControl_Handshake[8].Start := FALSE;
            // Action Qualifier=R
            // Token: "ST10_GeneralData".FlowControl_Handshake[8].Done
            "ST10_GeneralData".FlowControl_Handshake[8].Done := FALSE;

            // Transition to next step: 373
            IF TRUE THEN  // Sequential transition - review XML for actual condition
                #State := STEP_ST10_Flow8_FRobot_2_WaitGripperPos3ScanFinish;
            END_IF;

        // ===========================================
        // STEP 373: WaitGripperPos3ScanFinish
        // ===========================================
        STEP_ST10_Flow8_FRobot_2_WaitGripperPos3ScanFinish:
            // No actions in XML

            // Transition to next step: 296
            IF TRUE THEN  // Sequential transition - review XML for actual condition
                #State := STEP_ST10_Flow8_FRobot_2_WaitGripperPos1ScanFinish;
            END_IF;

        // ===========================================
        // STEP 296: WaitGripperPos1ScanFinish
        // ===========================================
        STEP_ST10_Flow8_FRobot_2_WaitGripperPos1ScanFinish:
            // No actions in XML

            // Transition to next step: 385
            IF TRUE THEN  // Sequential transition - review XML for actual condition
                #State := STEP_ST10_Flow8_FRobot_2_WaitGripperPos4ScanFinish;
            END_IF;

        // ===========================================
        // STEP 385: WaitGripperPos4ScanFinish
        // ===========================================
        STEP_ST10_Flow8_FRobot_2_WaitGripperPos4ScanFinish:
            // No actions in XML

            // Transition to next step: 900
            IF TRUE THEN  // Sequential transition - review XML for actual condition
                #State := STEP_ST10_Flow8_FRobot_2_S_900;
            END_IF;

        // ===========================================
        // STEP 900: 900
        // ===========================================
        STEP_ST10_Flow8_FRobot_2_S_900:
            // No actions in XML

            // Transition to next step: 249
            IF TRUE THEN  // Sequential transition - review XML for actual condition
                #State := STEP_ST10_Flow8_FRobot_2_PartOKStatus;
            END_IF;

        // ===========================================
        // STEP 249: PartOKStatus
        // ===========================================
        STEP_ST10_Flow8_FRobot_2_PartOKStatus:
            // Action Qualifier=N
            // Token: "AutoProcessData".F_Robot2Grip2.PartStatus := 199
            "AutoProcessData".F_Robot2Grip2.PartStatus := 199;

            // Transition to next step: 343
            IF TRUE THEN  // Sequential transition - review XML for actual condition
                #State := STEP_ST10_Flow8_FRobot_2_WaitRobotFinish_1;
            END_IF;

        // ===========================================
        // STEP 343: WaitRobotFinish_1
        // ===========================================
        STEP_ST10_Flow8_FRobot_2_WaitRobotFinish_1:
            // No actions in XML

            // Transition to next step: 369
            IF TRUE THEN  // Sequential transition - review XML for actual condition
                #State := STEP_ST10_Flow8_FRobot_2_WaitRobotGripStatus_3;
            END_IF;

        // ===========================================
        // STEP 369: WaitRobotGripStatus_3
        // ===========================================
        STEP_ST10_Flow8_FRobot_2_WaitRobotGripStatus_3:
            // No actions in XML

            // Transition to next step: 243
            IF TRUE THEN  // Sequential transition - review XML for actual condition
                #State := STEP_ST10_Flow8_FRobot_2_Grip1PartStatus;
            END_IF;

        // ===========================================
        // STEP 243: Grip1PartStatus
        // ===========================================
        STEP_ST10_Flow8_FRobot_2_Grip1PartStatus:
            // Action Qualifier=N
            // Token: "AutoProcessData".F_Robot2Grip2.PartStatus := 100
            "AutoProcessData".F_Robot2Grip2.PartStatus := 100;

            // Transition to next step: 301
            IF TRUE THEN  // Sequential transition - review XML for actual condition
                #State := STEP_ST10_Flow8_FRobot_2_RobotScanGripPos1Comp;
            END_IF;

        // ===========================================
        // STEP 301: RobotScanGripPos1Comp
        // ===========================================
        STEP_ST10_Flow8_FRobot_2_RobotScanGripPos1Comp:
            // No actions in XML

            // Transition to next step: 361
            IF TRUE THEN  // Sequential transition - review XML for actual condition
                #State := STEP_ST10_Flow8_FRobot_2_StartRobotPutPress;
            END_IF;

        // ===========================================
        // STEP 361: StartRobotPutPress
        // ===========================================
        STEP_ST10_Flow8_FRobot_2_StartRobotPutPress:
            // Action Qualifier=N
            // Token: "KukaRobot2_CtrlDB".sPLCtoROB.User.Cycle.DI273_PutPressReq
            "KukaRobot2_CtrlDB".sPLCtoROB.User.Cycle.DI273_PutPressReq;

            // Transition to next step: 706
            IF TRUE THEN  // Sequential transition - review XML for actual condition
                #State := STEP_ST10_Flow8_FRobot_2_WaitRobotHomeRequest;
            END_IF;

        // ===========================================
        // STEP 706: WaitRobotHomeRequest
        // ===========================================
        STEP_ST10_Flow8_FRobot_2_WaitRobotHomeRequest:
            // Action Qualifier=R
            // Token: "ChangeOver_DB".Robot_2.MaintenancePosReqSelFlag
            "ChangeOver_DB".Robot_2.MaintenancePosReqSelFlag := FALSE;

            // Transition to next step: 929
            IF TRUE THEN  // Sequential transition - review XML for actual condition
                #State := STEP_ST10_Flow8_FRobot_2_BrakeTestFinish;
            END_IF;

        // ===========================================
        // STEP 929: BrakeTestFinish
        // ===========================================
        STEP_ST10_Flow8_FRobot_2_BrakeTestFinish:
            // Action Qualifier=R
            // Token: "Robot_DB".Robot_2.BrakeTest_Req
            "Robot_DB".Robot_2.BrakeTest_Req := FALSE;

            // Transition to next step: 9
            IF TRUE THEN  // Sequential transition - review XML for actual condition
                #State := STEP_ST10_Flow8_FRobot_2_S9;
            END_IF;

        // ===========================================
        // STEP 9: S9
        // ===========================================
        STEP_ST10_Flow8_FRobot_2_S9:
            // No actions in XML

            // Transition to next step: 200
            IF TRUE THEN  // Sequential transition - review XML for actual condition
                #State := STEP_ST10_Flow8_FRobot_2_Tablecode_Scan;
            END_IF;

        // ===========================================
        // STEP 200: Tablecode Scan
        // ===========================================
        STEP_ST10_Flow8_FRobot_2_Tablecode_Scan:
            // Action Qualifier=R
            // Token: "KukaRobot2_CtrlDB".sPLCtoROB.User.Cycle.DI307_ScanPartFinish
            "KukaRobot2_CtrlDB".sPLCtoROB.User.Cycle.DI307_ScanPartFinish := FALSE;
            // Action Qualifier=R
            // Token: "KukaRobot2_CtrlDB".sPLCtoROB.User.Cycle.DI306_ScanPartComplete
            "KukaRobot2_CtrlDB".sPLCtoROB.User.Cycle.DI306_ScanPartComplete := FALSE;
            // Action Qualifier=N
            // Token: "AutoProcessData".GripperCode_R2[1] := ''
            "AutoProcessData".GripperCode_R2[1] := '';
            // Action Qualifier=N
            // Token: "AutoProcessData".GripperCode_R2[2] := ''
            "AutoProcessData".GripperCode_R2[2] := '';
            // Action Qualifier=N
            // Token: "AutoProcessData".GripperCode_R2[3] := ''
            "AutoProcessData".GripperCode_R2[3] := '';
            // Action Qualifier=N
            // Token: "AutoProcessData".GripperCode_R2[4] := ''
            "AutoProcessData".GripperCode_R2[4] := '';

            // Transition to next step: 328
            IF TRUE THEN  // Sequential transition - review XML for actual condition
                #State := STEP_ST10_Flow8_FRobot_2_StartRobotScanNGPut;
            END_IF;

        // ===========================================
        // STEP 328: StartRobotScanNGPut
        // ===========================================
        STEP_ST10_Flow8_FRobot_2_StartRobotScanNGPut:
            // Action Qualifier=N
            // Token: "KukaRobot2_CtrlDB".sPLCtoROB.User.Cycle.DI249_ScanNGPutReq
            "KukaRobot2_CtrlDB".sPLCtoROB.User.Cycle.DI249_ScanNGPutReq;

            // Transition to next step: 450
            IF TRUE THEN  // Sequential transition - review XML for actual condition
                #State := STEP_ST10_Flow8_FRobot_2_ScanMaganeProcess;
            END_IF;

        // ===========================================
        // STEP 450: ScanMaganeProcess
        // ===========================================
        STEP_ST10_Flow8_FRobot_2_ScanMaganeProcess:
            // No actions in XML

            // Transition to next step: 326
            IF TRUE THEN  // Sequential transition - review XML for actual condition
                #State := STEP_ST10_Flow8_FRobot_2_StartRobotPickPalletShaft;
            END_IF;

        // ===========================================
        // STEP 326: StartRobotPickPalletShaft
        // ===========================================
        STEP_ST10_Flow8_FRobot_2_StartRobotPickPalletShaft:
            // Action Qualifier=N
            // Token: "KukaRobot2_CtrlDB".sPLCtoROB.User.Cycle.DI241_PickPalletReq
            "KukaRobot2_CtrlDB".sPLCtoROB.User.Cycle.DI241_PickPalletReq;

            // Transition to next step: 356
            IF TRUE THEN  // Sequential transition - review XML for actual condition
                #State := STEP_ST10_Flow8_FRobot_2_WaitRobotFinish_4;
            END_IF;

        // ===========================================
        // STEP 356: WaitRobotFinish_4
        // ===========================================
        STEP_ST10_Flow8_FRobot_2_WaitRobotFinish_4:
            // Action Qualifier=N
            // Token: "KukaRobot2_CtrlDB".sPLCtoROB.User.Cycle.DI262_ScanPartComplete
            "KukaRobot2_CtrlDB".sPLCtoROB.User.Cycle.DI262_ScanPartComplete;

            // Transition to next step: 260
            IF TRUE THEN  // Sequential transition - review XML for actual condition
                #State := STEP_ST10_Flow8_FRobot_2_DataMove_3;
            END_IF;

        // ===========================================
        // STEP 260: DataMove_3
        // ===========================================
        STEP_ST10_Flow8_FRobot_2_DataMove_3:
            // Action Qualifier=N, Event="S1"
            // Token: "AutoProcessData".B_Press2 := "AutoProcessData".F_Robot2Grip1
            "AutoProcessData".B_Press2 := "AutoProcessData".F_Robot2Grip1;
            // Action Qualifier=N, Event="S1"
            // Token: "AutoProcessData".F_Robot2Grip1 := "AutoProcessData".ClearData
            "AutoProcessData".F_Robot2Grip1 := "AutoProcessData".ClearData;

            // Transition to next step: 499
            IF TRUE THEN  // Sequential transition - review XML for actual condition
                #State := STEP_ST10_Flow8_FRobot_2_ScanMaganeProcessFinish;
            END_IF;

        // ===========================================
        // STEP 499: ScanMaganeProcessFinish
        // ===========================================
        STEP_ST10_Flow8_FRobot_2_ScanMaganeProcessFinish:
            // Action Qualifier=S
            // Token: #ioPM_Inface.ProcessComplete
            #ioPM_Inface.ProcessComplete := TRUE;
            // Action Qualifier=R
            // Token: #ioPM_Inface.ProcessStart
            #ioPM_Inface.ProcessStart := FALSE;

            // Transition to next step: 120
            IF TRUE THEN  // Sequential transition - review XML for actual condition
                #State := STEP_ST10_Flow8_FRobot_2_ScanNGPut;
            END_IF;

        // ===========================================
        // STEP 120: ScanNGPut
        // ===========================================
        STEP_ST10_Flow8_FRobot_2_ScanNGPut:
            // Action Qualifier=S
            // Token: "AutoProcessControl".Robot_2.ScanNGPutFlag
            "AutoProcessControl".Robot_2.ScanNGPutFlag := TRUE;
            // Action Qualifier=R
            // Token: #ioPM_Inface.ProcessComplete
            #ioPM_Inface.ProcessComplete := FALSE;
            // Action Qualifier=S
            // Token: #ioPM_Inface.ProcessStart
            #ioPM_Inface.ProcessStart := TRUE;

            // Transition to next step: 347
            IF TRUE THEN  // Sequential transition - review XML for actual condition
                #State := STEP_ST10_Flow8_FRobot_2_WaitRobotGripHaveStatus_1;
            END_IF;

        // ===========================================
        // STEP 347: WaitRobotGripHaveStatus_1
        // ===========================================
        STEP_ST10_Flow8_FRobot_2_WaitRobotGripHaveStatus_1:
            // No actions in XML

            // Transition to next step: 264
            IF TRUE THEN  // Sequential transition - review XML for actual condition
                #State := STEP_ST10_Flow8_FRobot_2_DataMove_5;
            END_IF;

        // ===========================================
        // STEP 264: DataMove_5
        // ===========================================
        STEP_ST10_Flow8_FRobot_2_DataMove_5:
            // Action Qualifier=N
            // Token: "AutoProcessData".C_Glue.Code_1 := "AutoProcessData".F_Robot2Grip2.Code_1
            "AutoProcessData".C_Glue.Code_1 := "AutoProcessData".F_Robot2Grip2.Code_1;
            // Action Qualifier=N
            // Token: "AutoProcessData".C_Glue.PartStatus := 320
            "AutoProcessData".C_Glue.PartStatus := 320;

            // Transition to next step: 384
            IF TRUE THEN  // Sequential transition - review XML for actual condition
                #State := STEP_ST10_Flow8_FRobot_2_MES_Online__offline_;
            END_IF;

        // ===========================================
        // STEP 384: MES Online  offline?
        // ===========================================
        STEP_ST10_Flow8_FRobot_2_MES_Online__offline_:
            // No actions in XML

            // Transition to next step: 359
            IF TRUE THEN  // Sequential transition - review XML for actual condition
                #State := STEP_ST10_Flow8_FRobot_2_WaitRobotFinish_5;
            END_IF;

        // ===========================================
        // STEP 359: WaitRobotFinish_5
        // ===========================================
        STEP_ST10_Flow8_FRobot_2_WaitRobotFinish_5:
            // No actions in XML

            // Transition to next step: 246
            IF TRUE THEN  // Sequential transition - review XML for actual condition
                #State := STEP_ST10_Flow8_FRobot_2_ScanStart;
            END_IF;

        // ===========================================
        // STEP 246: ScanStart
        // ===========================================
        STEP_ST10_Flow8_FRobot_2_ScanStart:
            // Action Qualifier=S
            // Token: "KeyenceSR1000Ctrl_806A1DB".ioAutoTrigger
            "KeyenceSR1000Ctrl_806A1DB".ioAutoTrigger := TRUE;

            // Transition to next step: 251
            IF TRUE THEN  // Sequential transition - review XML for actual condition
                #State := STEP_ST10_Flow8_FRobot_2_PartNGStatus;
            END_IF;

        // ===========================================
        // STEP 251: PartNGStatus
        // ===========================================
        STEP_ST10_Flow8_FRobot_2_PartNGStatus:
            // Action Qualifier=N
            // Token: "AutoProcessData".F_Robot2Grip2.PartStatus := 155
            "AutoProcessData".F_Robot2Grip2.PartStatus := 155;

            // Transition to next step: 331
            IF TRUE THEN  // Sequential transition - review XML for actual condition
                #State := STEP_ST10_Flow8_FRobot_2_Gripe1StatusAlarm;
            END_IF;

        // ===========================================
        // STEP 331: Gripe1StatusAlarm
        // ===========================================
        STEP_ST10_Flow8_FRobot_2_Gripe1StatusAlarm:
            // Action Qualifier=S
            // Token: "ST10_DeviceError".F.Robot_2.Grip1Error
            "ST10_DeviceError".F.Robot_2.Grip1Error := TRUE;

            // Transition to next step: 245
            IF TRUE THEN  // Sequential transition - review XML for actual condition
                #State := STEP_ST10_Flow8_FRobot_2_CheckScanReady;
            END_IF;

        // ===========================================
        // STEP 245: CheckScanReady
        // ===========================================
        STEP_ST10_Flow8_FRobot_2_CheckScanReady:
            // No actions in XML

            // Transition to next step: 332
            IF TRUE THEN  // Sequential transition - review XML for actual condition
                #State := STEP_ST10_Flow8_FRobot_2_Gripe2StatusAlarm;
            END_IF;

        // ===========================================
        // STEP 332: Gripe2StatusAlarm
        // ===========================================
        STEP_ST10_Flow8_FRobot_2_Gripe2StatusAlarm:
            // Action Qualifier=S
            // Token: "ST10_DeviceError".F.Robot_2.Grip2Error
            "ST10_DeviceError".F.Robot_2.Grip2Error := TRUE;

            // Transition to next step: 110
            IF TRUE THEN  // Sequential transition - review XML for actual condition
                #State := STEP_ST10_Flow8_FRobot_2_ScanFixtureCode;
            END_IF;

        // ===========================================
        // STEP 110: ScanFixtureCode
        // ===========================================
        STEP_ST10_Flow8_FRobot_2_ScanFixtureCode:
            // Action Qualifier=R
            // Token: #ioPM_Inface.ProcessComplete
            #ioPM_Inface.ProcessComplete := FALSE;
            // Action Qualifier=S
            // Token: #ioPM_Inface.ProcessStart
            #ioPM_Inface.ProcessStart := TRUE;

            // Transition to next step: 346
            IF TRUE THEN  // Sequential transition - review XML for actual condition
                #State := STEP_ST10_Flow8_FRobot_2_WaitRobotGripHaveStatus;
            END_IF;

        // ===========================================
        // STEP 346: WaitRobotGripHaveStatus
        // ===========================================
        STEP_ST10_Flow8_FRobot_2_WaitRobotGripHaveStatus:
            // No actions in XML

            // Transition to next step: 345
            IF TRUE THEN  // Sequential transition - review XML for actual condition
                #State := STEP_ST10_Flow8_FRobot_2_WaitRobotFinish_2;
            END_IF;

        // ===========================================
        // STEP 345: WaitRobotFinish_2
        // ===========================================
        STEP_ST10_Flow8_FRobot_2_WaitRobotFinish_2:
            // No actions in XML

            // Transition to next step: 599
            IF TRUE THEN  // Sequential transition - review XML for actual condition
                #State := STEP_ST10_Flow8_FRobot_2_PutProcessFinish;
            END_IF;

        // ===========================================
        // STEP 599: PutProcessFinish
        // ===========================================
        STEP_ST10_Flow8_FRobot_2_PutProcessFinish:
            // Action Qualifier=S
            // Token: #ioPM_Inface.ProcessComplete
            #ioPM_Inface.ProcessComplete := TRUE;
            // Action Qualifier=R
            // Token: #ioPM_Inface.ProcessStart
            #ioPM_Inface.ProcessStart := FALSE;
            // Action Qualifier=N
            // Token: "Robot_DB".Robot_2.SpeedCount := "Robot_DB".Robot_2.SpeedCount + 1
            "Robot_DB".Robot_2.SpeedCount := "Robot_DB".Robot_2.SpeedCount + 1;

            // Transition to next step: 899
            IF TRUE THEN  // Sequential transition - review XML for actual condition
                #State := STEP_ST10_Flow8_FRobot_2_WaitR1HomePosFinsh_1;
            END_IF;

        // ===========================================
        // STEP 899: WaitR1HomePosFinsh_1
        // ===========================================
        STEP_ST10_Flow8_FRobot_2_WaitR1HomePosFinsh_1:
            // No actions in XML

            // Transition to next step: 125
            IF TRUE THEN  // Sequential transition - review XML for actual condition
                #State := STEP_ST10_Flow8_FRobot_2_GlueNGPut;
            END_IF;

        // ===========================================
        // STEP 125: GlueNGPut
        // ===========================================
        STEP_ST10_Flow8_FRobot_2_GlueNGPut:
            // Action Qualifier=S
            // Token: "AutoProcessControl".Robot_2.GlueNGPutFlag
            "AutoProcessControl".Robot_2.GlueNGPutFlag := TRUE;
            // Action Qualifier=R
            // Token: #ioPM_Inface.ProcessComplete
            #ioPM_Inface.ProcessComplete := FALSE;
            // Action Qualifier=S
            // Token: #ioPM_Inface.ProcessStart
            #ioPM_Inface.ProcessStart := TRUE;

            // Transition to next step: 253
            IF TRUE THEN  // Sequential transition - review XML for actual condition
                #State := STEP_ST10_Flow8_FRobot_2_DataMove;
            END_IF;

        // ===========================================
        // STEP 253: DataMove
        // ===========================================
        STEP_ST10_Flow8_FRobot_2_DataMove:
            // Action Qualifier=N, Event="S1"
            // Token: "AutoProcessData".C_MagnScanNGBuffer := "AutoProcessData".F_Robot2Grip2
            "AutoProcessData".C_MagnScanNGBuffer := "AutoProcessData".F_Robot2Grip2;
            // Action Qualifier=N, Event="S1"
            // Token: "AutoProcessData".F_Robot2Grip2 := "AutoProcessData".ClearData
            "AutoProcessData".F_Robot2Grip2 := "AutoProcessData".ClearData;

            // Transition to next step: 131
            IF TRUE THEN  // Sequential transition - review XML for actual condition
                #State := STEP_ST10_Flow8_FRobot_2_Maintenance;
            END_IF;

        // ===========================================
        // STEP 131: Maintenance
        // ===========================================
        STEP_ST10_Flow8_FRobot_2_Maintenance:
            // Action Qualifier=R
            // Token: #ioPM_Inface.ProcessComplete
            #ioPM_Inface.ProcessComplete := FALSE;
            // Action Qualifier=S
            // Token: #ioPM_Inface.ProcessStart
            #ioPM_Inface.ProcessStart := TRUE;

            // Transition to next step: 500
            IF TRUE THEN  // Sequential transition - review XML for actual condition
                #State := STEP_ST10_Flow8_FRobot_2_GluePickProcess;
            END_IF;

        // ===========================================
        // STEP 500: GluePickProcess
        // ===========================================
        STEP_ST10_Flow8_FRobot_2_GluePickProcess:
            // No actions in XML

            // Transition to next step: 336
            IF TRUE THEN  // Sequential transition - review XML for actual condition
                #State := STEP_ST10_Flow8_FRobot_2_SetGripCodeScanFlag;
            END_IF;

        // ===========================================
        // STEP 336: SetGripCodeScanFlag
        // ===========================================
        STEP_ST10_Flow8_FRobot_2_SetGripCodeScanFlag:
            // No actions in XML

            // Transition to next step: 704
            IF TRUE THEN  // Sequential transition - review XML for actual condition
                #State := STEP_ST10_Flow8_FRobot_2_ReqRobotToMantenPos_1;
            END_IF;

        // ===========================================
        // STEP 704: ReqRobotToMantenPos_1
        // ===========================================
        STEP_ST10_Flow8_FRobot_2_ReqRobotToMantenPos_1:
            // Action Qualifier=N
            // Token: "KukaRobot2_CtrlDB".sPLCtoROB.User.Cycle.DI297_MaintainRequest
            "KukaRobot2_CtrlDB".sPLCtoROB.User.Cycle.DI297_MaintainRequest;

            // Transition to next step: 357
            IF TRUE THEN  // Sequential transition - review XML for actual condition
                #State := STEP_ST10_Flow8_FRobot_2_WaitRobotReachScanPos;
            END_IF;

        // ===========================================
        // STEP 357: WaitRobotReachScanPos
        // ===========================================
        STEP_ST10_Flow8_FRobot_2_WaitRobotReachScanPos:
            // No actions in XML

            // Transition to next step: 399
            IF TRUE THEN  // Sequential transition - review XML for actual condition
                #State := STEP_ST10_Flow8_FRobot_2_GlueNGPutFinish;
            END_IF;

        // ===========================================
        // STEP 399: GlueNGPutFinish
        // ===========================================
        STEP_ST10_Flow8_FRobot_2_GlueNGPutFinish:
            // Action Qualifier=S
            // Token: #ioPM_Inface.ProcessComplete
            #ioPM_Inface.ProcessComplete := TRUE;
            // Action Qualifier=R
            // Token: #ioPM_Inface.ProcessStart
            #ioPM_Inface.ProcessStart := FALSE;

            // Transition to next step: 449
            IF TRUE THEN  // Sequential transition - review XML for actual condition
                #State := STEP_ST10_Flow8_FRobot_2_PickTableProcessFinish;
            END_IF;

        // ===========================================
        // STEP 449: PickTableProcessFinish
        // ===========================================
        STEP_ST10_Flow8_FRobot_2_PickTableProcessFinish:
            // Action Qualifier=S
            // Token: #ioPM_Inface.ProcessComplete
            #ioPM_Inface.ProcessComplete := TRUE;
            // Action Qualifier=R
            // Token: #ioPM_Inface.ProcessStart
            #ioPM_Inface.ProcessStart := FALSE;

            // Transition to next step: 910
            IF TRUE THEN  // Sequential transition - review XML for actual condition
                #State := STEP_ST10_Flow8_FRobot_2_MasteringTest_Req;
            END_IF;

        // ===========================================
        // STEP 910: MasteringTest_Req
        // ===========================================
        STEP_ST10_Flow8_FRobot_2_MasteringTest_Req:
            // Action Qualifier=N
            // Token: "KukaRobot2_CtrlDB".sPLCtoROB.User.Cycle.DI321
            "KukaRobot2_CtrlDB".sPLCtoROB.User.Cycle.DI321;
            // Action Qualifier=N
            // Token: "KukaRobot2_CtrlDB".sPLCtoROB.User.Safety.DI450
            "KukaRobot2_CtrlDB".sPLCtoROB.User.Safety.DI450;

            // Transition to next step: 338
            IF TRUE THEN  // Sequential transition - review XML for actual condition
                #State := STEP_ST10_Flow8_FRobot_2_StartRobotScanGripperCode;
            END_IF;

        // ===========================================
        // STEP 338: StartRobotScanGripperCode
        // ===========================================
        STEP_ST10_Flow8_FRobot_2_StartRobotScanGripperCode:
            // Action Qualifier=N
            // Token: "KukaRobot2_CtrlDB".sPLCtoROB.User.Cycle.DI305_GripScan
            "KukaRobot2_CtrlDB".sPLCtoROB.User.Cycle.DI305_GripScan;

            // Transition to next step: 340
            IF TRUE THEN  // Sequential transition - review XML for actual condition
                #State := STEP_ST10_Flow8_FRobot_2_RobotScanGripperReachPos1;
            END_IF;

        // ===========================================
        // STEP 340: RobotScanGripperReachPos1
        // ===========================================
        STEP_ST10_Flow8_FRobot_2_RobotScanGripperReachPos1:
            // No actions in XML

            // Transition to next step: 911
            IF TRUE THEN  // Sequential transition - review XML for actual condition
                #State := STEP_ST10_Flow8_FRobot_2_WaitMasteringTestFinish;
            END_IF;

        // ===========================================
        // STEP 911: WaitMasteringTestFinish
        // ===========================================
        STEP_ST10_Flow8_FRobot_2_WaitMasteringTestFinish:
            // No actions in XML

            // Transition to next step: 360
            IF TRUE THEN  // Sequential transition - review XML for actual condition
                #State := STEP_ST10_Flow8_FRobot_2_WaitRobotGripStatus;
            END_IF;

        // ===========================================
        // STEP 360: WaitRobotGripStatus
        // ===========================================
        STEP_ST10_Flow8_FRobot_2_WaitRobotGripStatus:
            // No actions in XML

            // Transition to next step: 3
            IF TRUE THEN  // Sequential transition - review XML for actual condition
                #State := STEP_ST10_Flow8_FRobot_2_S3;
            END_IF;

        // ===========================================
        // STEP 3: S3
        // ===========================================
        STEP_ST10_Flow8_FRobot_2_S3:
            // No actions in XML

            // Transition to next step: 299
            IF TRUE THEN  // Sequential transition - review XML for actual condition
                #State := STEP_ST10_Flow8_FRobot_2_PickPalletFinish;
            END_IF;

        // ===========================================
        // STEP 299: PickPalletFinish
        // ===========================================
        STEP_ST10_Flow8_FRobot_2_PickPalletFinish:
            // Action Qualifier=S
            // Token: #ioPM_Inface.ProcessComplete
            #ioPM_Inface.ProcessComplete := TRUE;
            // Action Qualifier=R
            // Token: #ioPM_Inface.ProcessStart
            #ioPM_Inface.ProcessStart := FALSE;

            // Transition to next step: 550
            IF TRUE THEN  // Sequential transition - review XML for actual condition
                #State := STEP_ST10_Flow8_FRobot_2_PutPressProcess;
            END_IF;

        // ===========================================
        // STEP 550: PutPressProcess
        // ===========================================
        STEP_ST10_Flow8_FRobot_2_PutPressProcess:
            // No actions in XML

            // Transition to next step: 266
            IF TRUE THEN  // Sequential transition - review XML for actual condition
                #State := STEP_ST10_Flow8_FRobot_2_Grip1SensorError;
            END_IF;

        // ===========================================
        // STEP 266: Grip1SensorError
        // ===========================================
        STEP_ST10_Flow8_FRobot_2_Grip1SensorError:
            // Action Qualifier=S
            // Token: "ST10_DeviceError".F.Robot_2.Grip1SensorCheckError
            "ST10_DeviceError".F.Robot_2.Grip1SensorCheckError := TRUE;

            // Transition to next step: 600
            IF TRUE THEN  // Sequential transition - review XML for actual condition
                #State := STEP_ST10_Flow8_FRobot_2_PressPickProcess;
            END_IF;

        // ===========================================
        // STEP 600: PressPickProcess
        // ===========================================
        STEP_ST10_Flow8_FRobot_2_PressPickProcess:
            // No actions in XML

            // Transition to next step: 265
            IF TRUE THEN  // Sequential transition - review XML for actual condition
                #State := STEP_ST10_Flow8_FRobot_2_Data_Clear_6;
            END_IF;

        // ===========================================
        // STEP 265: Data Clear_6
        // ===========================================
        STEP_ST10_Flow8_FRobot_2_Data_Clear_6:
            // Action Qualifier=N, Event="S1"
            // Token: "AutoProcessData".F_Robot2Grip2 := "AutoProcessData".ClearData
            "AutoProcessData".F_Robot2Grip2 := "AutoProcessData".ClearData;

            // Transition to next step: 355
            IF TRUE THEN  // Sequential transition - review XML for actual condition
                #State := STEP_ST10_Flow8_FRobot_2_StartRobotScanRing;
            END_IF;

        // ===========================================
        // STEP 355: StartRobotScanRing
        // ===========================================
        STEP_ST10_Flow8_FRobot_2_StartRobotScanRing:
            // Action Qualifier=N
            // Token: "KukaRobot2_CtrlDB".sPLCtoROB.User.Cycle.DI261_ScanPartReq
            "KukaRobot2_CtrlDB".sPLCtoROB.User.Cycle.DI261_ScanPartReq;

            // Transition to next step: 327
            IF TRUE THEN  // Sequential transition - review XML for actual condition
                #State := STEP_ST10_Flow8_FRobot_2_WaitRobotFinish;
            END_IF;

        // ===========================================
        // STEP 327: WaitRobotFinish
        // ===========================================
        STEP_ST10_Flow8_FRobot_2_WaitRobotFinish:
            // No actions in XML

            // Transition to next step: 333
            IF TRUE THEN  // Sequential transition - review XML for actual condition
                #State := STEP_ST10_Flow8_FRobot_2_RobotTaskSelect;
            END_IF;

        // ===========================================
        // STEP 333: RobotTaskSelect
        // ===========================================
        STEP_ST10_Flow8_FRobot_2_RobotTaskSelect:
            // No actions in XML

            // Transition to next step: 149
            IF TRUE THEN  // Sequential transition - review XML for actual condition
                #State := STEP_ST10_Flow8_FRobot_2_Tablecode_ScanFinish;
            END_IF;

        // ===========================================
        // STEP 149: Tablecode ScanFinish
        // ===========================================
        STEP_ST10_Flow8_FRobot_2_Tablecode_ScanFinish:
            // Action Qualifier=S
            // Token: #ioPM_Inface.ProcessComplete
            #ioPM_Inface.ProcessComplete := TRUE;
            // Action Qualifier=R
            // Token: #ioPM_Inface.ProcessStart
            #ioPM_Inface.ProcessStart := FALSE;

            // Transition to next step: 330
            IF TRUE THEN  // Sequential transition - review XML for actual condition
                #State := STEP_ST10_Flow8_FRobot_2_GripStatusCheck;
            END_IF;

        // ===========================================
        // STEP 330: GripStatusCheck
        // ===========================================
        STEP_ST10_Flow8_FRobot_2_GripStatusCheck:
            // No actions in XML

            // Transition to next step: 368
            IF TRUE THEN  // Sequential transition - review XML for actual condition
                #State := STEP_ST10_Flow8_FRobot_2_WaitRobotFinish_8;
            END_IF;

        // ===========================================
        // STEP 368: WaitRobotFinish_8
        // ===========================================
        STEP_ST10_Flow8_FRobot_2_WaitRobotFinish_8:
            // No actions in XML

            // Transition to next step: 365
            IF TRUE THEN  // Sequential transition - review XML for actual condition
                #State := STEP_ST10_Flow8_FRobot_2_WaitRobotFinish_7;
            END_IF;

        // ===========================================
        // STEP 365: WaitRobotFinish_7
        // ===========================================
        STEP_ST10_Flow8_FRobot_2_WaitRobotFinish_7:
            // No actions in XML

            // Transition to next step: 364
            IF TRUE THEN  // Sequential transition - review XML for actual condition
                #State := STEP_ST10_Flow8_FRobot_2_StartRobotPressPick;
            END_IF;

        // ===========================================
        // STEP 364: StartRobotPressPick
        // ===========================================
        STEP_ST10_Flow8_FRobot_2_StartRobotPressPick:
            // No actions in XML

            // Transition to next step: 705
            IF TRUE THEN  // Sequential transition - review XML for actual condition
                #State := STEP_ST10_Flow8_FRobot_2_WaitR1MaintenPosFinsh_1;
            END_IF;

        // ===========================================
        // STEP 705: WaitR1MaintenPosFinsh_1
        // ===========================================
        STEP_ST10_Flow8_FRobot_2_WaitR1MaintenPosFinsh_1:
            // Action Qualifier=R
            // Token: "AutoProcessControl".Robot_2.MaintenanceRequest
            "AutoProcessControl".Robot_2.MaintenanceRequest := FALSE;

            // Transition to next step: 130
            IF TRUE THEN  // Sequential transition - review XML for actual condition
                #State := STEP_ST10_Flow8_FRobot_2_PickTable;
            END_IF;

        // ===========================================
        // STEP 130: PickTable
        // ===========================================
        STEP_ST10_Flow8_FRobot_2_PickTable:
            // Action Qualifier=R
            // Token: #ioPM_Inface.ProcessComplete
            #ioPM_Inface.ProcessComplete := FALSE;
            // Action Qualifier=S
            // Token: #ioPM_Inface.ProcessStart
            #ioPM_Inface.ProcessStart := TRUE;

            // Transition to next step: 311
            IF TRUE THEN  // Sequential transition - review XML for actual condition
                #State := STEP_ST10_Flow8_FRobot_2_RobotReady_;
            END_IF;

        // ===========================================
        // STEP 311: RobotReady?
        // ===========================================
        STEP_ST10_Flow8_FRobot_2_RobotReady_:
            // No actions in XML

            // Transition to next step: 132
            IF TRUE THEN  // Sequential transition - review XML for actual condition
                #State := STEP_ST10_Flow8_FRobot_2_Masref_test;
            END_IF;

        // ===========================================
        // STEP 132: Masref_test
        // ===========================================
        STEP_ST10_Flow8_FRobot_2_Masref_test:
            // Action Qualifier=R
            // Token: #ioPM_Inface.ProcessComplete
            #ioPM_Inface.ProcessComplete := FALSE;
            // Action Qualifier=S
            // Token: #ioPM_Inface.ProcessStart
            #ioPM_Inface.ProcessStart := TRUE;

            // Transition to next step: 650
            IF TRUE THEN  // Sequential transition - review XML for actual condition
                #State := STEP_ST10_Flow8_FRobot_2_GluePutProcess;
            END_IF;

        // ===========================================
        // STEP 650: GluePutProcess
        // ===========================================
        STEP_ST10_Flow8_FRobot_2_GluePutProcess:
            // No actions in XML

            // Transition to next step: 358
            IF TRUE THEN  // Sequential transition - review XML for actual condition
                #State := STEP_ST10_Flow8_FRobot_2_StartRobotGluePick;
            END_IF;

        // ===========================================
        // STEP 358: StartRobotGluePick
        // ===========================================
        STEP_ST10_Flow8_FRobot_2_StartRobotGluePick:
            // Action Qualifier=N
            // Token: "KukaRobot2_CtrlDB".sPLCtoROB.User.Cycle.DI269_GluePickReq
            "KukaRobot2_CtrlDB".sPLCtoROB.User.Cycle.DI269_GluePickReq;

            // Transition to next step: 649
            IF TRUE THEN  // Sequential transition - review XML for actual condition
                #State := STEP_ST10_Flow8_FRobot_2_PressPickProcessFinish_;
            END_IF;

        // ===========================================
        // STEP 649: PressPickProcessFinish_
        // ===========================================
        STEP_ST10_Flow8_FRobot_2_PressPickProcessFinish_:
            // Action Qualifier=S
            // Token: #ioPM_Inface.ProcessComplete
            #ioPM_Inface.ProcessComplete := TRUE;
            // Action Qualifier=R
            // Token: #ioPM_Inface.ProcessStart
            #ioPM_Inface.ProcessStart := FALSE;

            // Transition to next step: 707
            IF TRUE THEN  // Sequential transition - review XML for actual condition
                #State := STEP_ST10_Flow8_FRobot_2_ReqRobotToHomePos;
            END_IF;

        // ===========================================
        // STEP 707: ReqRobotToHomePos
        // ===========================================
        STEP_ST10_Flow8_FRobot_2_ReqRobotToHomePos:
            // Action Qualifier=N
            // Token: "KukaRobot2_CtrlDB".sPLCtoROB.User.Cycle.DI300_HomeRequest
            "KukaRobot2_CtrlDB".sPLCtoROB.User.Cycle.DI300_HomeRequest;

            // Transition to next step: 252
            IF TRUE THEN  // Sequential transition - review XML for actual condition
                #State := STEP_ST10_Flow8_FRobot_2_DataClear;
            END_IF;

        // ===========================================
        // STEP 252: DataClear
        // ===========================================
        STEP_ST10_Flow8_FRobot_2_DataClear:
            // Action Qualifier=N, Event="S1"
            // Token: "AutoProcessData".F_Robot2Grip2 := "AutoProcessData".ClearData
            "AutoProcessData".F_Robot2Grip2 := "AutoProcessData".ClearData;

            // Transition to next step: 352
            IF TRUE THEN  // Sequential transition - review XML for actual condition
                #State := STEP_ST10_Flow8_FRobot_2_StartRobotPickTable;
            END_IF;

        // ===========================================
        // STEP 352: StartRobotPickTable
        // ===========================================
        STEP_ST10_Flow8_FRobot_2_StartRobotPickTable:
            // Action Qualifier=N
            // Token: "KukaRobot2_CtrlDB".sPLCtoROB.User.Cycle.DI257_PickPartReq
            "KukaRobot2_CtrlDB".sPLCtoROB.User.Cycle.DI257_PickPartReq;

            // Transition to next step: 381
            IF TRUE THEN  // Sequential transition - review XML for actual condition
                #State := STEP_ST10_Flow8_FRobot_2_WaitRobotStartHome;
            END_IF;

        // ===========================================
        // STEP 381: WaitRobotStartHome
        // ===========================================
        STEP_ST10_Flow8_FRobot_2_WaitRobotStartHome:
            // No actions in XML

            // Transition to next step: 699
            IF TRUE THEN  // Sequential transition - review XML for actual condition
                #State := STEP_ST10_Flow8_FRobot_2_GluePutProcessFinish;
            END_IF;

        // ===========================================
        // STEP 699: GluePutProcessFinish
        // ===========================================
        STEP_ST10_Flow8_FRobot_2_GluePutProcessFinish:
            // Action Qualifier=S
            // Token: #ioPM_Inface.ProcessComplete
            #ioPM_Inface.ProcessComplete := TRUE;
            // Action Qualifier=R
            // Token: #ioPM_Inface.ProcessStart
            #ioPM_Inface.ProcessStart := FALSE;

            // Transition to next step: 363
            IF TRUE THEN  // Sequential transition - review XML for actual condition
                #State := STEP_ST10_Flow8_FRobot_2_WaitRobotGripStatus_1;
            END_IF;

        // ===========================================
        // STEP 363: WaitRobotGripStatus_1
        // ===========================================
        STEP_ST10_Flow8_FRobot_2_WaitRobotGripStatus_1:
            // No actions in XML

            // Transition to next step: 362
            IF TRUE THEN  // Sequential transition - review XML for actual condition
                #State := STEP_ST10_Flow8_FRobot_2_WaitRobotFinish_6;
            END_IF;

        // ===========================================
        // STEP 362: WaitRobotFinish_6
        // ===========================================
        STEP_ST10_Flow8_FRobot_2_WaitRobotFinish_6:
            // No actions in XML

            // Transition to next step: 250
            IF TRUE THEN  // Sequential transition - review XML for actual condition
                #State := STEP_ST10_Flow8_FRobot_2_PickPalletProcess;
            END_IF;

        // ===========================================
        // STEP 250: PickPalletProcess
        // ===========================================
        STEP_ST10_Flow8_FRobot_2_PickPalletProcess:
            // No actions in XML

            // Transition to next step: 4
            IF TRUE THEN  // Sequential transition - review XML for actual condition
                #State := STEP_ST10_Flow8_FRobot_2_RobotSpeed;
            END_IF;

        // ===========================================
        // STEP 4: RobotSpeed
        // ===========================================
        STEP_ST10_Flow8_FRobot_2_RobotSpeed:
            // Action Qualifier=N
            // Token: "KukaRobot2_CtrlDB".iSpeedValue := 20
            "KukaRobot2_CtrlDB".iSpeedValue := 20;

            // Transition to next step: 382
            IF TRUE THEN  // Sequential transition - review XML for actual condition
                #State := STEP_ST10_Flow8_FRobot_2_RobotManuallyMoved_;
            END_IF;

        // ===========================================
        // STEP 382: RobotManuallyMoved?
        // ===========================================
        STEP_ST10_Flow8_FRobot_2_RobotManuallyMoved_:
            // No actions in XML

            // Transition to next step: 257
            IF TRUE THEN  // Sequential transition - review XML for actual condition
                #State := STEP_ST10_Flow8_FRobot_2_DataMove_2;
            END_IF;

        // ===========================================
        // STEP 257: DataMove_2
        // ===========================================
        STEP_ST10_Flow8_FRobot_2_DataMove_2:
            // Action Qualifier=N, Event="S1"
            // Token: "AutoProcessData".F_Robot2Grip1 := "AutoProcessData".C_Glue
            "AutoProcessData".F_Robot2Grip1 := "AutoProcessData".C_Glue;
            // Action Qualifier=N, Event="S1"
            // Token: "AutoProcessData".C_Glue := "AutoProcessData".ClearData
            "AutoProcessData".C_Glue := "AutoProcessData".ClearData;

            // Transition to next step: 267
            IF TRUE THEN  // Sequential transition - review XML for actual condition
                #State := STEP_ST10_Flow8_FRobot_2_Grip2SensorError;
            END_IF;

        // ===========================================
        // STEP 267: Grip2SensorError
        // ===========================================
        STEP_ST10_Flow8_FRobot_2_Grip2SensorError:
            // Action Qualifier=S
            // Token: "ST10_DeviceError".F.Robot_2.Grip2SensorCheckError
            "ST10_DeviceError".F.Robot_2.Grip2SensorCheckError := TRUE;

            // Transition to next step: 921
            IF TRUE THEN  // Sequential transition - review XML for actual condition
                #State := STEP_ST10_Flow8_FRobot_2_WaitBrakeTestFinish;
            END_IF;

        // ===========================================
        // STEP 921: WaitBrakeTestFinish
        // ===========================================
        STEP_ST10_Flow8_FRobot_2_WaitBrakeTestFinish:
            // No actions in XML

            // Transition to next step: 268
            IF TRUE THEN  // Sequential transition - review XML for actual condition
                #State := STEP_ST10_Flow8_FRobot_2_FlagReset;
            END_IF;

        // ===========================================
        // STEP 268: FlagReset
        // ===========================================
        STEP_ST10_Flow8_FRobot_2_FlagReset:
            // Action Qualifier=R
            // Token: "AutoProcessControl".Robot_2.PalletPickFlag
            "AutoProcessControl".Robot_2.PalletPickFlag := FALSE;
            // Action Qualifier=R
            // Token: "AutoProcessControl".Robot_2.MagnetScanFlag
            "AutoProcessControl".Robot_2.MagnetScanFlag := FALSE;
            // Action Qualifier=R
            // Token: "AutoProcessControl".Robot_2.GluePutFlag
            "AutoProcessControl".Robot_2.GluePutFlag := FALSE;
            // Action Qualifier=R
            // Token: "AutoProcessControl".Robot_2.GluePickFlag
            "AutoProcessControl".Robot_2.GluePickFlag := FALSE;
            // Action Qualifier=R
            // Token: "AutoProcessControl".Robot_2.Press2PutFlag
            "AutoProcessControl".Robot_2.Press2PutFlag := FALSE;
            // Action Qualifier=R
            // Token: "AutoProcessControl".Robot_2.GlueNGPutFlag
            "AutoProcessControl".Robot_2.GlueNGPutFlag := FALSE;
            // Action Qualifier=R
            // Token: "AutoProcessControl".Robot_2.ScanNGPutFlag
            "AutoProcessControl".Robot_2.ScanNGPutFlag := FALSE;

            // Transition to next step: 150
            IF TRUE THEN  // Sequential transition - review XML for actual condition
                #State := STEP_ST10_Flow8_FRobot_2_PressPick;
            END_IF;

        // ===========================================
        // STEP 150: PressPick
        // ===========================================
        STEP_ST10_Flow8_FRobot_2_PressPick:
            // Action Qualifier=R
            // Token: #ioPM_Inface.ProcessComplete
            #ioPM_Inface.ProcessComplete := FALSE;
            // Action Qualifier=S
            // Token: #ioPM_Inface.ProcessStart
            #ioPM_Inface.ProcessStart := TRUE;

            // Transition to next step: 337
            IF TRUE THEN  // Sequential transition - review XML for actual condition
                #State := STEP_ST10_Flow8_FRobot_2_WaitGripperPos2ScanFinish;
            END_IF;

        // ===========================================
        // STEP 337: WaitGripperPos2ScanFinish
        // ===========================================
        STEP_ST10_Flow8_FRobot_2_WaitGripperPos2ScanFinish:
            // No actions in XML

            // Transition to next step: 378
            IF TRUE THEN  // Sequential transition - review XML for actual condition
                #State := STEP_ST10_Flow8_FRobot_2_RobotScanGripPos3Comp;
            END_IF;

        // ===========================================
        // STEP 378: RobotScanGripPos3Comp
        // ===========================================
        STEP_ST10_Flow8_FRobot_2_RobotScanGripPos3Comp:
            // No actions in XML

            // Transition to next step: 919
            IF TRUE THEN  // Sequential transition - review XML for actual condition
                #State := STEP_ST10_Flow8_FRobot_2_MasteringTestFinish;
            END_IF;

        // ===========================================
        // STEP 919: MasteringTestFinish
        // ===========================================
        STEP_ST10_Flow8_FRobot_2_MasteringTestFinish:
            // Action Qualifier=R
            // Token: "Robot_DB".Robot_2.MasteringTest_Req
            "Robot_DB".Robot_2.MasteringTest_Req := FALSE;

    END_CASE;

    // UPDATE ioPM_Inface
    #ioPM_Inface.InitialRun := #act_InitialRun;
    #ioPM_Inface.InitialOK := #act_InitialOK;
    #ioPM_Inface.WaitRunning := #act_WaitRunning;
    #ioPM_Inface.Running := #act_Running;
    #ioPM_Inface.ProcessComplete := #act_ProcessComplete;
    #ioPM_Inface.ProcessStart := #act_ProcessStart;
    #ioPM_Inface.UnPause := #act_UnPause;

    // ERROR HANDLING
    IF #bError THEN
        #ioStatus := 900;
        #oAlarmID := INT_TO_WORD(#wErrorID);
    ELSE
        #ioStatus := 0;
        #oAlarmID := 0;
    END_IF;
END_FUNCTION_BLOCK

//=============================================================================
// END OF FILE
//=============================================================================
